{attribute 'GeneratedUsingTerminal: ELX9560-0000-0018'}
{attribute addProperty BoxType "ELX9560-0000-0018"}
{attribute addProperty Id "Uex_OKAT %I*BOOL1"}
{attribute addProperty CRC "2203005008"}
{attribute addProperty Size "1"}
TYPE Status_Uex_834F3050 :
STRUCT
	{attribute addProperty Name "Uex_OK"}
	Uex_OK AT %I* : BOOL;
END_STRUCT
END_TYPE

(* stored: Version 1.2.0.0, ProductVersion 3.1.4024.9
   DUT Status_Uex_834F3050: Id {07b41074-9fc7-4b31-937b-2f04495c9432} *)
